FUNCTION_BLOCK GrundstrukturSkill IMPLEMENTS I_State_Skill
VAR_INPUT
	bExecute			:BOOL;				// Trigger für Ausführung von Skill
	iSysCommand			:eSystemCommand;	// Steuerungsvariabel von System (Resetten)
	iObjState			:eObjectState;		// Information über Zustand von Objekt
	iSysState			:eSystemState;		// Information über Zustand von System
END_VAR
VAR_OUTPUT
	iSkillCommand		:eSkillCommand;		// Steuerungsvariable für Anlagenmodell
	bDone				:BOOL;				// Information ob Skill ausgfeührt wurde
	bBusy				:BOOL;				// Information ob Skill im Moment ausgeführt wird
	bLimit				:BOOL;				// Information ob Skill an einem Limit angekommen ist
	bError				:BOOL;				// Information ob sich Skill in Fehlerzustand befindet
	iErrorID			:INT;				// Information um welchen Fehler es sich handelt
END_VAR
VAR
	// Managementvariablen
	iState				:eSkillState;		// Information über Zustand von Skill
	bTargetReached		:BOOL;				// Information ob Prozessziel erreicht wurde
	bLimitReached		:BOOL;				// Information ob Limit erreicht wurde
	
	// Startvariablen (FB soll nur bei einer steigenden Flanke gestartet werden)
	fTrigger			:R_TRIG;			// Erkennung einer steigenden Flanke für den Starte
	fSwitch				:SR;				// Setzen des Signals
	bSwitchResett		:BOOL;				// Resetten des Signals
	
	// Zustandsvariablen
	bStarten			:BOOL;
	bStoppen			:BOOL;
	bObjektFertig		:BOOL;
	bWertErreicht		:BOOL;				
	bLimitErreicht		:BOOL;				
	bSkillFertig		:BOOL;
	bFehler				:BOOL;
	bResetten			:BOOL;
	
	
END_VAR

PROPERTY P_State : eSkillState
GET
P_State := iState;
END_GET
END_PROPERTY

END_FUNCTION_BLOCK

(* stored: Version 1.1.0.1
   POU GrundstrukturSkill: Id {8849c73d-5d94-464c-8fa0-5cada18e040f}, SpecialFunc None
   Property P_State: Id {174b5214-bae6-4f3c-b2eb-b050fc2deeb8}
   Get Get: Id {611af6d0-4b12-4b33-98af-b90cc15ee0fa} *)
